FUNCTION_BLOCK L1_MCEmitter (* Layer 1 multicast emitter *)
  (* Standard: 61499-2 *)
  (* Version 0.0, 2015-03-03, EQUEROL, UJI *)
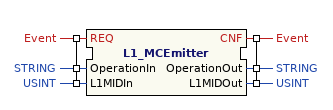
  EVENT_INPUT
    REQ WITH OperationIn, L1MIDIn; (* Request multicast send to all blocks in layer 1 *)
  END_EVENT
  EVENT_OUTPUT
    CNF WITH OperationOut, L1MIDOut; (* Multicast emission *)
  END_EVENT
  VAR_INPUT
    OperationIn : STRING; (* Serialized operation *)
    L1MIDIn : USINT; (* Layer 1 multicast identifier *)
  END_VAR
  VAR_OUTPUT
    OperationOut : STRING; (* Serialized operation *)
    L1MIDOut : USINT; (* Layer 1 multicast identifier *)
  END_VAR
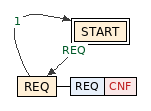
  EC_STATES
    START; (* Initial State *)
    REQ : REQ -> CNF; (* Normal execution *)
  END_STATES
  EC_TRANSITIONS
    START TO REQ := REQ;
    REQ TO START := 1;
  END_TRANSITIONS
  ALGORITHM REQ IN ST: (* Normally executed algorithm *)
OperationIn := OperationOut;
L1MIDIn := L1MIDOut;
  END_ALGORITHM
END_FUNCTION_BLOCK
